# EPICS autosave request: soft_iocs/galil_DMC_E04/iocBoot/iocgalil_DMC_E04/slit_settings.req
file "2slit_soft_settings.req", P=$(P), SLIT=XenocsUS_V:
file "2slit_soft_settings.req", P=$(P), SLIT=XenocsUS_H:
file "2slit_soft_settings.req", P=$(P), SLIT=XenocsDS_V:
file "2slit_soft_settings.req", P=$(P), SLIT=XenocsDS_H:
